Staubli VAL3: page_instr.pjx

--- page_instr.pjx ---
Parameters version=s7.7 stackSize=5000 millimeterUnit=true
Program file=buildList.pgx
Program file=goTo.pgx
Program file=listAdd.pgx
Program file=loadPage.pgx
Program file=loadTemplate.pgx
Program file=main.pgx
Program file=onBackEvent.pgx
Program file=onEnterEvent.pgx
Program file=onExit.pgx
Program file=onF1Event.pgx
Program file=onF2Event.pgx
Program file=onF3Event.pgx
Program file=onF4Event.pgx
Program file=onF5Event.pgx
Program file=onF6Event.pgx
Program file=onF7Event.pgx
Program file=onF8Event.pgx
Program file=onStart.pgx
Program file=refresh.pgx
Program file=refreshDynamic.pgx
Program file=refreshStatic.pgx
Program file=saveIt.pgx
Data file=page_instr.dtx
Library alias=page path=Disk://kernel/template/page/page.pjx
Library alias=use path=Disk://kernel/userPage/userPage.pjx
Library alias=language path=Disk://kernel/language/language.pjx
Library alias=saveData path=Disk://saveData/saveData.pjx
Library alias=events path=Disk://..//templates/instruction/instruction.pjx
Library alias=prog path=Disk://instruction/PROG/PROG.pjx
Library alias=cycleStatus path=Disk://cycleStatus/cycleStatus.pjx
Library alias=TrajItem path=Disk://../templates/trajectory/trajectory.pjx
Library alias=sub path=Disk://instruction/SUB/SUB.pjx
Library alias=saveInputOutput path=Disk://saveInputOutput/saveInputOutput.pjx
Library alias=tcp path=Disk://kernel/tool/tool.pjx
Type name=InstrItem path=Disk://kernel/template/InstrItem/InstrItem.pjx
Type name=TrajectoryItem path=Disk://kernel/template/TrajectoryItem/TrajectoryItem.pjx
Type name=progItem path=Disk://kernel/template/progItem/progItem.pjx
Type name=dioItem path=Disk://kernel/template/dioItem/dioItem.pjx

--- page_instr.dtx ---
num nIndex
num nIndexItem = 1
num nKey = 255
public num nPage
num nRefresh = 2571.459
num nSelected
num nTime = 1
num nView
num nViewItem = 1
string sEvent = " 1 OUT valve1>ON"
string sField[2]
  [0] = "Disk://trajectory/PALLET/page_pallet"
  [1] = "hello"
public string sItems = "test"
string sList = " 1 OUT valve1>ON"
string sMenu[8]
  [2] = "I/O"
  [3] = "Paste"
  [4] = "Mark"
  [5] = "Delete"
  [6] = "Insert"
  [7] = "Save"
string sMenu8[8]
string sMessage
string sProgram = "test"
bool bButton[8]
  [1] = true
  [2] = true
  [3] = true
  [4] = true
  [5] = true
  [6] = true
  [7] = true
bool bExit = true
bool bLarge
num nId
bool bMoveRelease
num nOldIndex
string sPath

--- main.pgx ---
public program main()
  local bool l_bSave
  local num l_nIndex
  local string l_sEvent
  local bool l_bFound
  local InstrItem l_iInstr
  local string l_sPath
  local bool l_bUnreached
  local string l_sMessage
begin
  // INIT
  call onStart()
  // LOOP UNTIL nKey=255
  do
    // refresh
    call refresh()
    nKey=getKey()
    call use:listevent(nKey,nId,sEvent)
    nSelected=nId
    nView=use:nView
    // get the index
    if find(left(sEvent,1)," ")!=-1
      l_sEvent=right(sEvent,len(sEvent)-1)
    else
      l_sEvent=sEvent
    endIf
    toNum(l_sEvent,l_nIndex,l_bFound)
    if l_bFound
      nIndex=l_nIndex-1
    endIf
    // check for the moveHold
    call prog:getItem(l_iInstr,nIndex)
    call saveData:getPathInstr(l_iInstr.sType,l_sPath)
    if find(l_sPath,"trajectory")!=-1
      call goTo(l_bUnreached,l_iInstr)
      if l_bUnreached
        // show the message out of range
        call language:message(l_sMessage,-5)
        call use:timerDialog(l_sMessage,1)
        l_bUnreached=false
      endIf
    endIf
    // key capture
    switch nKey
      case 259
        // TAB-> ENLARGE
        bLarge=!bLarge
        call use:setView(bLarge)
      break
      case 263
        // backSpace
        if l_bFound
          call onBackEvent(l_bSave)
        endIf
      break
      case 271
        // Simulation
        if l_bFound
          call onF1Event()
        endIf
      break
      case 272
        call onF2Event(l_bSave)
      break
      case 273
        // INPUT OUTPUT
        call onF3Event(l_bSave)
      break
      case 274
        // PASTE
        call onF4Event(l_bSave)
      break
      case 275
        // SELECT_UNSELECT
        if l_bFound
          call onF5Event()
        endIf
      break
      case 276
        // DELETE
        if l_bFound
          call onF6Event(l_bSave)
        endIf
      break
      case 277
        //INSERT
        if l_bFound or l_sEvent==""
          call onF7Event(l_bSave)
        endIf
      break
      case 278
        // SAVE
        call onF8Event(l_bSave)
      break
      case 270
        if l_bFound
          // EDIT THE FIELD
          call onEnterEvent(l_bSave)
        endIf
      break
      case 255
        // exit??
        // on Exit
        call onExit(l_bSave)
      break
    endSwitch
    //release the resource
    delay(0.1)
  until bExit
  //
  // reset
  //
  bExit=false
end

--- buildList.pgx ---
program buildList()
  local num l_nSize
  local InstrItem l_iEvent
  local num i
  local string l_sEmpty
  local num l_nResult
  local num l_nSizeItem
  local num j
  local TrajectoryItem l_tTraj
  local string l_sPath
  local num k
  local progItem l_pProg
  local string l_sData
  local string l_sType
begin
  // INIT the list
  l_sEmpty=""
  call use:stringCopy(l_sEmpty,sList)
  // add the items
  call prog:getSizeItem(l_nSize)
  for i=0 to (l_nSize-1)
    call prog:getItem(l_iEvent,i)
    if l_iEvent.sType!=""
      l_sData=l_iEvent.sData
      l_sType=l_iEvent.sType
      call saveInputOutput:replaceIO(l_sData,l_sType,l_sData)
      call listAdd(toString("2",i+1)+" "+l_sType+" "+l_sData)
      if find(l_iEvent.sType,"#")!=-1
        l_iEvent.sType=right(l_iEvent.sType,len(l_iEvent.sType)-1)
      endIf
      // show the name of IN OUT NUM
      if saveData:bShowItem and find(l_iEvent.sData,"@")==-1
        // get inside the trajectory field
        call saveData:getPathInstr(l_iEvent.sType,l_sPath)
        // TRAJECTORY
        if TrajItem:libLoad(l_sPath)==0
          delay(0)
          // scan for the action
          call TrajItem:load(l_iEvent.sData,l_nResult)
          if l_nResult==0
            call TrajItem:getSizeItem(false,l_nSizeItem)
            // patch for the PALLET
            if find(TrajItem:libPath(),"PALLET")!=-1
              l_nSizeItem=1
            endIf
            // scan for the TCP
            for j=0 to l_nSizeItem-1
              call TrajItem:getTrajItem(l_tTraj,j)
              // scan for the TCP
              if l_tTraj.nTcpAction==1
                call listAdd("  -TCP ON ")
              elseIf l_tTraj.nTcpAction==2
                call listAdd("  -TCP OFF ")
              endIf
              for k=0 to size(l_tTraj.iInstr)-1
                if l_tTraj.iInstr[k].sType!=""
                  l_sData=l_tTraj.iInstr[k].sData
                  l_sType=l_tTraj.iInstr[k].sType
                  call saveInputOutput:replaceIO(l_sData,l_sType,l_sData)
                  call listAdd("   -"+l_sType+" "+l_sData)
                endIf
              endFor
            endFor
          endIf
        elseIf l_iEvent.sType=="SUB"
          // SUB
          call sub:load(l_iEvent.sData,l_nResult)
          if l_nResult==0
            call sub:getProgItem(l_pProg,l_iEvent.sData)
            l_nSizeItem=size(l_pProg.iEvent)
            for j=0 to l_nSizeItem-1
              if l_pProg.iEvent[j].sType!=""
                l_sData=l_pProg.iEvent[j].sData
                l_sType=l_pProg.iEvent[j].sType
                call saveInputOutput:replaceIO(l_sData,l_sType,l_sData)
                call listAdd("  -"+l_sType+" "+l_sData)
              endIf
            endFor
          endIf
        endIf
      endIf
    else
      // delete empty space
      call prog:deleteItem(i,l_nResult)
      // recovery
      call prog:getSizeItem(l_nSize)
      i=i-1
    endIf
  endFor
  //
  use:bUseRefresh=true
end

--- goTo.pgx ---
program goTo(bool& x_bUnreached[], InstrItem x_iInstrItem)
  local bool l_bUnreached
  local num l_nIndexTool
  local tool l_tTool
  local num l_nSize
  local string l_sItems[2]
  local num l_nId
  local num l_nResult
  local TrajectoryItem l_tTraj
  local string l_sPath
  local num l_nIndex
begin
//  // check the cycle status
//  if !cycleStatus:bCycle and !cycleStatus:bSimulation
//    // check the working Mode
//    if cycleStatus:nWorkingMode==1 and isPowered()
//      // set the memory for the moveHold button
//      if cycleStatus:nWorkingStatus==6
//        bMoveRelease=true
//      endIf
//      // check for the index
//      if nOldIndex!=l_nIndex or (cycleStatus:nWorkingStatus!=0 and cycleStatus:nWorkingStatus!=6)
//        if !isEmpty()
//          resetMotion()
//        endIf
//        if nOldIndex!=l_nIndex
//          nOldIndex=l_nIndex
//        endIf
//      else
//        if isEmpty() and cycleStatus:nWorkingStatus==0 and bMoveRelease
//          bMoveRelease=false
//          cls()
//          // copy the item to the trajectory
//          l_sItems=x_iInstrItem.sData
//          // take the elements
//          call saveData:getPathInstr(x_iInstrItem.sType,l_sPath)
//          if l_sPath!=sPath
//            sPath=l_sPath
//            TrajItem:libLoad(l_sPath)
//          endIf
//          call TrajItem:load(l_sItems,l_nResult)
//          call TrajItem:getSizeItem(false,l_nSize)
//          // MOVE
//          do
//            if l_nIndex>0
//              call use:typeMenu(7,"<<")
//            else
//              call use:typeMenu(7,"    ")
//            endIf
//            if l_nIndex<=l_nSize
//              call use:typeMenu(8,">>")
//            else
//              call use:typeMenu(8,"    ")
//            endIf
//            // get the data to move
//            call TrajItem:getTool(l_nIndexTool)
//            call tcp:getTool(l_tTool,l_nIndexTool)
//            call TrajItem:getTrajItem(l_tTraj,l_nIndex)
//            //
//            // use a sTemp mdesc to set the blend off
//            //
//            l_tTraj.nom_speed.blend=off
//            call TrajItem:goTo(l_tTool,l_tTraj.nom_speed,l_tTraj.moveType,x_bUnreached,l_nIndex)
//            // TO DO language
//            call use:timerDialog("Going to point: "+toString("",l_nIndex+1)+ " / "+toString("",l_nSize),0)
//            do
//              l_nId=getKey()
//              call use:scroll(0,7,38,(getMoveId()-roundDown(getMoveId()))*100)
//              delay(0)
//            until isEmpty()or l_nId==255 or l_nId==277 or l_nId==278
//            // continue
//            if isEmpty() or (l_nId==278 and l_nIndex<l_nSize)
//              if isEmpty()
//                call use:timerDialog("At point: "+toString("",l_nIndex+1)+ " / "+toString("",l_nSize),1)
//              endIf
//              l_nIndex=l_nIndex+1
//            elseIf l_nId==277 and l_nIndex>0
//              // decrease
//              l_nIndex=l_nIndex-1
//            else
//              delay(1)
//            endIf
//            // release
//            resetMotion()
//          until x_bUnreached or l_nId==255 or l_nIndex>=l_nSize or(l_nIndex==l_nSize and l_nSize==1)
//          // refresh
//          use:bUseRefresh=true
//        endIf
//      endIf
//    else
//      // reset the cycle
//      if cycleStatus:nWorkingMode!=1 or !isPowered()
//        resetMotion()
//      endIf
//    endIf
//  endIf
//  if l_nId==255
//    // release
//    call use:nullKey(l_nId)
//  endIf
end

--- loadPage.pgx ---
program loadPage(string x_sPage, string& x_sItems[])
// load the next page
  local num i
  local string l_sMessage
begin
  // look if the page libload is correct
  i=page:libLoad(x_sPage)
  delay(0)
  if i!=0
    logMsg("[KERNEL] INTERFACE:PAGE LIBLOAD "+x_sPage+" result "+toString("",i))
    call language:message(l_sMessage,-7)
    popUpMsg(l_sMessage+x_sPage+" ; "+toString("",i))
  else
    // copy all the field from x_sItems to the next page
    call use:stringCopy(x_sItems,page:sItems)
    call page:main()
  endIf
end

--- loadTemplate.pgx ---
program loadTemplate()
begin
  // load the default instruction
  events:libLoad("Disk://..//templates/instruction")
  delay(0)
end

--- onBackEvent.pgx ---
program onBackEvent(bool& x_bSave[])
  local num i
  local string l_sItem
  local string l_sInstruction
  local num l_nIndex
  local num j
  local num l_nChar
  local num l_nResult
  local InstrItem l_iInstr
  local string l_sPath
begin
  //
  // NB sEvent is the selected
  // element in the LIST
  //
  // get the item
  call prog:getItem(l_iInstr,nIndex)
  // find the instruction to load
  call saveData:getPathInstr(l_iInstr.sType,l_sPath)
  j=events:libLoad(l_sPath)
  delay(0)
  if j==0
    // cal the onInsert function
    call events:onInsert(l_iInstr.sData)
    // insert the item
    if l_iInstr.sData!=""
      call prog:insertItem(l_iInstr,nIndex)
      if nIndex>0
        call prog:deleteItem(nIndex+1,l_nResult)
      endIf
      x_bSave=true
      logMsg("[KERNEL] INTERFACE:Insert new item: "+l_sItem)
      i=size(saveData:sInstr)-1
    endIf
    call buildList()
    //
  else
    popUpMsg("Loading event "+l_sInstruction+" error CODE "+toString("",j))
  endIf
  //
end

--- onEnterEvent.pgx ---
program onEnterEvent(bool& x_bSave[])
  local num i
  local string l_sInstruction
  local num j
  local num l_nDefault
  local bool l_bYes
  local bool l_bCancel
  local string l_sButton[2]
  local string l_sMessage
  local InstrItem l_iInstr
  local string l_sPath
  local num l_nResult
  local string l_sProgType
  local num l_nIndex
  local num l_nSelect
  local string l_sProgram
begin
  //
  // NB sEvent is the selected
  // element in the LIST
  //
  // get the item
  l_sProgType=saveData:sProgTypeUsing
  l_nIndex=nIndex
  l_nSelect=nSelected
  l_sProgram=sProgram
  call prog:getItem(l_iInstr,nIndex)
  call saveData:getPathInstr(l_iInstr.sType,l_sPath)
  // libload the instruction
  j=events:libLoad(l_sPath)
  delay(0)
  if j==0
    call prog:getItem(l_iInstr,nIndex)
    // copy
    sField=l_iInstr.sData
    call events:onEdit(sField)
    // reload the template
    call loadTemplate()
    //
    if find(sField,"Disk://")!=-1
      //
      // ask if you want to save yor modification
      //
      if x_bSave
        call language:message(l_sMessage,-1)
        // get the yes_no button Key
        call language:getYesNo(l_sButton)
        // ask the question
        call use:yes_no_cancel(l_sMessage,l_sButton,l_bYes,l_bCancel)
        if l_bYes
          call saveIt(x_bSave)
        endIf
      endIf
      // check if the cancel button has been pressed
      if !l_bCancel
        //
        // load the page
        //
        call loadPage(sField,sField[1])
        //
        // came back
        //
        if saveData:sProgTypeUsing!=l_sProgType or sField[1]!=l_sProgram
          // rebuild all
          saveData:sProgTypeUsing=l_sProgType
          nIndex=l_nIndex
          nSelected=l_nSelect
          sProgram=l_sProgram
          // load the program TYPE
          call saveData:getPathInstr(saveData:sProgTypeUsing,l_sPath)
          l_nResult=prog:libLoad(l_sPath)
          delay(0)
          // load the program
          call prog:load(sProgram,i)
          call refresh()
        endIf
      endIf
    else
      if l_iInstr.sData!=sField and !use:bUseEscape and l_iInstr.sData!=""
        // paste
        l_iInstr.sData=sField
        x_bSave=true
      endIf
      // look if every is OK
      call prog:setItem(l_iInstr,nIndex)
    endIf
    // rebuilt
    call buildList()
  else
    popUpMsg("Loading event "+l_iInstr.sType+" error CODE "+toString("",j))
  endIf
  // refresh
  use:bUseRefresh=true
end

--- onExit.pgx ---
program onExit(bool& x_bSave[])
  local string l_sMessage
  local bool l_bYes
  local bool l_bCancel
  local string l_sButton[2]
begin
  //
  // saveIt
  //
  if x_bSave
    call language:message(l_sMessage,-1)
    // get the yes_no button Key
    call language:getYesNo(l_sButton)
    // ask the question
    call use:yes_no_cancel(l_sMessage,l_sButton,l_bYes,l_bCancel)
    if l_bYes
      call saveIt(x_bSave)
    endIf
    // quit if not cancel
    bExit=!l_bCancel
  else
    // exit
    bExit=true
  endIf
end

--- onF1Event.pgx ---
program onF1Event()
  local bool l_bYes
  local string l_sMessage
  local string l_sItem
  local string l_sButton[2]
  local string l_sPage
  local InstrItem l_iItem
begin
  // look if the bButton is enable
  if bButton[0]
    //
    //
    // the SIMULATION is disable when cycle is active
    //
    if !cycleStatus:bCycle and find(left(sEvent,5),"-")==-1
      call language:message(l_sMessage,214)
      // get the yes_no button Key
      call language:getYesNo(l_sButton)
      // ask the question
      call use:yes_no(l_sMessage,l_sButton,l_bYes)
      if l_bYes
        call prog:getItem(l_iItem,nIndex)
        cycleStatus:iToSuperV=l_iItem
        cycleStatus:nInterfaceToSV=3
        logMsg("[KERNEL] INTERFACE:Simulation of the item: "+sEvent)
        wait(cycleStatus:nInterfaceToSV==-1)
        // load the production page
        l_sPage="simulation"
        call loadPage("kernel/page/production",l_sPage)
        call use:setView(false)
      endIf
    endIf
  endIf
end

--- onF2Event.pgx ---
program onF2Event(bool& x_bSave[])
  local string l_sEvent
  local num l_nIndex
  local num i
  local num l_nActualProg
  local string l_sMessage
  local string l_sButton[2]
  local bool l_bYes
  local string l_sResult
  local string l_sItem
  local string l_sEmpty
begin
  // look if the bButton is enable
  if bButton[1]
    // none
  endIf
end

--- onF3Event.pgx ---
program onF3Event(bool& x_bSave[])
  local string l_sMessage
  local num l_nActualProg
  local string l_sButton[2]
  local bool l_bYes
  local bool l_bCancel
  local string l_sEmpty
  local num i
begin
  // look if the bButton is enable
  if bButton[2]
    if x_bSave
      call language:message(l_sMessage,-1)
      // get the yes_no button Key
      call language:getYesNo(l_sButton)
      // ask the question
      call use:yes_no_cancel(l_sMessage,l_sButton,l_bYes,l_bCancel)
      if l_bYes
        call saveIt(x_bSave)
      endIf
    endIf
    // check if the cancel button has been pressed
    if !l_bCancel
      l_sEmpty=""
      call loadPage("Disk://instruction/inputOutput/page_inOut",l_sEmpty)
      call prog:load(sProgram,i)
      if i!=0
        // show the error message
        call language:message(l_sMessage,-7)
        popUpMsg(l_sMessage+" PROG "+sProgram+", "+toString("",i))
      endIf
      // return to the page
      logMsg("[KERNEL] INTERFACE:Page Edit Program: "+sProgram)
      call buildList()
    endIf
  endIf
end

--- onF4Event.pgx ---
program onF4Event(bool& x_bSave[])
begin
  // look if the bButton is enable
  if bButton[3]
    // paste the items select
    call prog:pasteItem(nIndex)
    logMsg("[KERNEL] INTERFACE:Paste progs items")
    call buildList()
    x_bSave=true
  endIf
end

--- onF5Event.pgx ---
program onF5Event()
  local num l_nSize
begin
  // look if the bButton is enable
  if bButton[4]
    //
    // select/ unselect the items
    //
    call prog:selectItem(nIndex)
    call prog:getSizeItem(l_nSize)
    // go down
    if nIndex<l_nSize-1
      nSelected=nId+1
    endIf
    call buildList()
  endIf
end

--- onF6Event.pgx ---
program onF6Event(bool& l_bSave[])
  local bool l_bYes
  local string l_sMessage
  local string l_sButton[2]
  local num l_nResult
begin
  // look if the bButton is enable
  if bButton[5]
    //
    // Delete the select Item
    //
    call language:message(l_sMessage,80)
    // get the yes_no button Key
    call language:getYesNo(l_sButton)
    // ask the question
    call use:yes_no(l_sMessage,l_sButton,l_bYes)
    if l_bYes
      call prog:deleteItem(nIndex,l_nResult)
      // go back by one
      if nIndex>0
        nSelected=nId-1
      endIf
      call buildList()
      l_bSave=true
    endIf
  endIf
end

--- onF7Event.pgx ---
program onF7Event(bool& x_bSave[])
  local num l_nIndex
  local string l_sItem
  local num i
  local num l_nResult
  local string l_sMessage
  local string l_sOrigin
  local string l_sPath
  local InstrItem l_iItem
begin
  // look if the bButton is enable
  if bButton[6]
    //
    //
    // insert a new field
    //
    if nIndex<0 or sEvent==""
      l_nIndex=0
    else
      //
      // insert a new field after
      //
      l_nIndex=nIndex+1
    endIf
    // show the list
    call use:setSizeList(14,0,12,11)
    call use:setView(false)
    call use:listcreate("")
    call use:clear(0,13)
    call language:message(l_sMessage,66)
    call use:type(0,13,l_sMessage)
    if saveData:sProgTypeUsing=="PROG"
      call use:listadd(saveData:sInstr)
    elseIf saveData:sProgTypeUsing=="SUB"
      // remove
      for i=0 to size(saveData:sInstrOnPoint)-1
        l_sItem=saveData:sInstrOnPoint[i]
        if l_sItem!="SUB"
          call use:listadd(l_sItem)
        endIf
      endFor
    endIf
    // update with the last select
    use:nView=nViewItem
    call use:listupdate(nIndexItem-nViewItem)
    l_sItem=""
    do
      i=get()
      call use:listevent(i,nIndexItem,l_sItem)
    until i==255 or i==270
    nViewItem=use:nView
    l_iItem.sType=l_sItem
    //
    // load the instruction
    if l_sItem!="" and i==270
      call saveData:getPathInstr(l_sItem,l_sPath)
      l_nResult=events:libLoad(l_sPath)
      delay(0)
      if l_nResult==0
        //
        call events:onInsert(l_iItem.sData)
        use:bUseEscape=false
        // insert the item
        if l_iItem.sData!=""
          call prog:insertItem(l_iItem,l_nIndex)
          nSelected=nSelected+1
          x_bSave=true
          logMsg("[KERNEL] INTERFACE:Insert new item: "+l_sItem)
          i=size(saveData:sInstr)-1
        endIf
      else
        logMsg("[KERNEL] INTERFACE:Error loading "+l_sItem+" error "+toString("",l_nResult))
      endIf
    endIf
    // rebuild the list
    use:nView=nView
    call buildList()
    call loadTemplate()
  endIf
  call use:nullKey(nKey)
end

--- onF8Event.pgx ---
program onF8Event(bool& l_bSave[])
  local num x_nResult
begin
  // look if the bButton is enable
  if bButton[7]
    //
    call saveIt(l_bSave)
  endIf
end

--- onStart.pgx ---
program onStart()
  local num i
  local string l_sMessage
  local string l_sPath
  local num l_nResult
begin
  // INIT
  sPath=""
  bExit=false
  nIndex=nSelected=nView=nId=0
  // reset the Key pressure
  call use:nullKey(nKey)
  // logMsg
  logMsg("[KERNEL] INTERFACE:PAGE edit program")
  // load the program TYPE
  call saveData:getPathInstr(saveData:sProgTypeUsing,l_sPath)
  l_nResult=prog:libLoad(l_sPath)
  delay(0)
  // program name
  sProgram=sItems[0]
  call prog:load(sProgram,i)
  //
  if i!=0
    call language:message(l_sMessage,-7)
    popUpMsg(l_sMessage+" PROG "+sProgram+" code "+toString("",i))
  endIf
  // unselect ALL
  call prog:unSelectItem()
  // define the list
  call buildList()
  // build the page
  call refreshStatic()
end

--- refreshStatic.pgx ---
program refreshStatic()
  local string l_sMessage
  local num l_nSize
  local string l_sEvent
  local num i
  local bool l_bType
begin
  cls()
  //
  // set the view of the page..
  //
  // SET THE PAGE NUMBER
  use:nPage=1000
  // USE <>PROFILE for <>PAGE
  use:nPage=use:nPage+abs(limit(saveData:mode,0,2)-2)
  if cycleStatus:bCycle
    use:nPage=use:nPage+3
  endIf
  // load the menu page
  if saveData:language!="japanese"
    // SET THE VIEW OF THE PAGE
    call language:page(l_sMessage,use:nPage)
    l_bType=true
    // define the menu
    call use:stringToArray(l_sMessage,sMenu)
  else
    // japanese use the array for the menu
    call language:page(sMenu8,use:nPage)
    l_bType=false
    call use:stringCopy(sMenu8,sMenu)
  endIf
  //
  call use:setMenu(sMenu,l_bType,3)
  call use:getMenu(sMenu,bButton)
  bButton[1]=true
  //
  // CREATE THE LIST
  //
  // define your list size for default
  call use:setSizeList(19,0,19,11)
  call use:setView(bLarge)
  //
  call use:listcreate(saveData:sProgTypeUsing+" "+sProgram)
  call use:listadd(sList)
  //
  // refresh
  call use:selectNewField(nSelected,nId,nView)
  nSelected=-1
end

--- saveIt.pgx ---
program saveIt(bool& x_bSave[])
  local string l_sMessage
  local num l_nResult
  local num l_nType
  local string l_sPath
begin
  // unselect ALL
  call prog:unSelectItem()
  // save
  call prog:save(sProgram,l_nResult)
  if l_nResult==0
    logMsg("[KERNEL] INTERFACE:Save the program: "+sProgram)
    x_bSave=false
    call language:message(l_sMessage,-4)
    call use:timerDialog(l_sMessage,1)
  else
    popUpMsg("Save code error "+toString("",l_nResult))
  endIf
end
